# EPICS autosave request: measCompApp/Db/measCompWaveformGenN_settings.req
$(P)$(R)Enable
$(P)$(R)Type
$(P)$(R)PulseWidth
$(P)$(R)PulseDelay
$(P)$(R)Amplitude
$(P)$(R)Offset
